// TIA Portal V20 export
DATA_BLOCK "ScaraArm3D"   // DB17, Motion_DB
// stored: InstanceOfName TO_Kinematics, OfSystemLibElement TO_Kinematics, OfSystemLibVersion 9.0
TO_Kinematics   // technology object, version 9.0
// stored: KinematicsAxis Ref J1_SCARA_Arm3D, Type TO_PositioningAxis, Index 1
// stored: KinematicsAxis Ref J3_SCARA_Arm3D, Type TO_PositioningAxis, Index 2
// stored: KinematicsAxis Ref J2_SCARA_Arm3D, Type TO_PositioningAxis, Index 3
// stored: KinematicsAxis Ref J4_SCARA_Arm3D, Type TO_PositioningAxis, Index 4
   // // inherited from TO_Object
   // VAR
   //    Tcp { ExternalWritable := 'False'; S7_SetPoint := 'True'} : TO_Struct_Kinematics_StatusKinematicsFrameTcp;
   //    Kinematics { S7_SetPoint := 'True'} : TO_Struct_Kinematics_Kinematics;
   //    KcsFrame { S7_SetPoint := 'True'} : TO_Struct_Kinematics_Frame;
   //    OcsFrame { S7_SetPoint := 'True'} : Array[1..3] of TO_Struct_Kinematics_Frame;
   //    Tool { S7_SetPoint := 'True'} : Array[1..3] of TO_Struct_Kinematics_Tool;
   //    DynamicDefaults { S7_SetPoint := 'True'} : TO_Struct_Kinematics_DynamicDefaults;
   //    DynamicLimits { S7_SetPoint := 'True'} : TO_Struct_Kinematics_DynamicLimits;
   //    Joint { S7_SetPoint := 'True'} : TO_Struct_Kinematics_Joint;
   //    AxisCoupling { S7_SetPoint := 'True'} : TO_Struct_Kinematics_AxisCoupling;
   //    MotionQueue { ExternalWritable := 'False'; S7_SetPoint := 'True'} : TO_Struct_Kinematics_MotionQueue;
   //    Transition { S7_SetPoint := 'True'} : TO_Struct_Kinematics_Transition;
   //    Override { S7_SetPoint := 'True'} : TO_Struct_Kinematics_Override;
   //    Conveyor { S7_SetPoint := 'True'} : TO_Struct_Kinematics_Conveyor;
   //    WorkspaceZone { S7_SetPoint := 'True'} : Array[1..10] of TO_Struct_Kinematics_WorkSpaceZone;
   //    KinematicsZone { S7_SetPoint := 'True'} : Array[2..10] of TO_Struct_Kinematics_KinematicsZone;
   //    StatusPath { ExternalWritable := 'False'; S7_SetPoint := 'True'} : TO_Struct_Kinematics_StatusPath;
   //    TcpInWcs { ExternalWritable := 'False'; S7_SetPoint := 'True'} : TO_Struct_Kinematics_StatusKinematicsFrameWithDynamics;
   //    TcpInOcs { ExternalWritable := 'False'; S7_SetPoint := 'True'} : Array[1..3] of TO_Struct_Kinematics_StatusKinematicsFrameWithDynamicsOcs;
   //    StatusOcsFrame { ExternalWritable := 'False'; S7_SetPoint := 'True'} : Array[1..3] of TO_Struct_Kinematics_StatusFrame;
   //    StatusKinematics { ExternalWritable := 'False'; S7_SetPoint := 'True'} : TO_Struct_Kinematics_StatusKinematics;
   //    AxesData { ExternalWritable := 'False'; S7_SetPoint := 'True'} : TO_Struct_Kinematics_AxesData;
   //    JointData { ExternalWritable := 'False'; S7_SetPoint := 'True'} : TO_Struct_Kinematics_StatusJointData;
   //    FlangeInKcs { ExternalWritable := 'False'; S7_SetPoint := 'True'} : TO_Struct_Kinematics_StatusFlangeInKcs;
   //    StatusTool { ExternalWritable := 'False'; S7_SetPoint := 'True'} : TO_Struct_Kinematics_StatusTool;
   //    StatusConveyor { ExternalWritable := 'False'; S7_SetPoint := 'True'} : Array[1..3] of TO_Struct_Kinematics_StatusConveyor;
   //    StatusWorkspaceZone { ExternalWritable := 'False'; S7_SetPoint := 'True'} : Array[1..10] of TO_Struct_Kinematics_StatusWorkSpaceZone;
   //    StatusKinematicsZone { ExternalWritable := 'False'; S7_SetPoint := 'True'} : Array[2..10] of TO_Struct_Kinematics_StatusKinematicsZone;
   //    StatusZoneMonitoring { ExternalWritable := 'False'; S7_SetPoint := 'True'} : TO_Struct_Kinematics_StatusZoneMonitoring;
   //    StatusMotionQueue { ExternalWritable := 'False'; S7_SetPoint := 'True'} : TO_Struct_Kinematics_StatusMotionQueue;
   //    KinematicsAxis { ExternalWritable := 'False'; S7_SetPoint := 'True'} : TO_Struct_Kinematics_KinematicsAxis;
   //    Units { ExternalWritable := 'False'; S7_SetPoint := 'True'} : TO_Struct_Kinematics_Units;
   //    StatusInterpreterMotion { ExternalWritable := 'False'; S7_SetPoint := 'True'} : TO_Struct_Kinematics_StatusInterpreterMotion;
   //    StatusWord { ExternalWritable := 'False'} : DWord;
   //    ErrorWord { ExternalWritable := 'False'} : DWord;
   //    ErrorDetail { ExternalWritable := 'False'; S7_SetPoint := 'True'} : TO_Struct_ErrorDetail;
   //    WarningWord { ExternalWritable := 'False'} : DWord;
   //    ControlPanel { S7_SetPoint := 'True'} : TO_Struct_Kinematics_ControlPanel;
   //    InternalToTrace { S7_SetPoint := 'True'} : Array[1..4] of TO_Struct_Internal;
   // END_VAR
BEGIN
   Kinematics.TypeOfKinematics := 10;
   Kinematics.Parameter[1] := 1028.48;
   Kinematics.Parameter[2] := 1150.0;
   Kinematics.Parameter[5] := 1200.0;
   Kinematics.Parameter[9..32] := 0.0;
   KcsFrame.x := 0.0;
   KcsFrame.y := 0.0;
   KcsFrame.z := 0.0;
   KcsFrame."a" := 0.0;
   KcsFrame."b" := 0.0;
   KcsFrame.c := 0.0;
   OcsFrame[2..3].x := 0.0;
   OcsFrame[2..3].y := 0.0;
   OcsFrame[2..3].z := 0.0;
   OcsFrame[2..3]."a" := 0.0;
   OcsFrame[1..3]."b" := 0.0;
   OcsFrame[1..3].c := 0.0;
   Tool[2..3].Frame.x := 0.0;
   Tool[2..3].Frame.y := 0.0;
   Tool[1].Frame.z := 50.0;
   Tool[2..3].Frame.z := 0.0;
   Tool[1..3].Frame."a" := 0.0;
   DynamicDefaults.Path.Velocity := 2000.0;
   DynamicDefaults.Path.Acceleration := 10000.0;
   DynamicDefaults.Path.Deceleration := 10000.0;
   DynamicDefaults.Path.Jerk := 100000.0;
   DynamicDefaults.Orientation.Velocity := 2000.0;
   DynamicDefaults.Orientation.Acceleration := 20000.0;
   DynamicDefaults.Orientation.Deceleration := 20000.0;
   DynamicDefaults.Orientation.Jerk := 1000000.0;
   DynamicDefaults.DynamicAdaption := 1;
   DynamicDefaults.MoveDirect.VelocityFactor := 0.5;
   DynamicDefaults.MoveDirect.AccelerationFactor := 0.5;
   DynamicDefaults.MoveDirect.DecelerationFactor := 0.5;
   DynamicDefaults.MoveDirect.JerkFactor := 0.5;
   DynamicLimits.Path.Velocity := 3000.0;
   DynamicLimits.Path.Acceleration := 100000.0;
   DynamicLimits.Path.Deceleration := 100000.0;
   DynamicLimits.Orientation.Velocity := 2200.0;
   DynamicLimits.Orientation.Acceleration := 20000.0;
   DynamicLimits.Orientation.Deceleration := 20000.0;
   DynamicLimits.Orientation.Jerk := 1000000.0;
   Override.Velocity := 62.0;
   WorkspaceZone[1].Active := true;
   WorkspaceZone[2..10].Active := false;
   WorkspaceZone[1].Valid := true;
   WorkspaceZone[2..10].Valid := false;
   WorkspaceZone[2..10]."Type" := 1;
   WorkspaceZone[1..10].ReferenceSystem := 0;
   WorkspaceZone[2..10].Frame.x := 0.0;
   WorkspaceZone[2..10].Frame.y := 0.0;
   WorkspaceZone[1].Frame.z := -100.0;
   WorkspaceZone[2..10].Frame.z := 0.0;
   WorkspaceZone[1..10].Frame."a" := 0.0;
   WorkspaceZone[1..10].Frame."b" := 0.0;
   WorkspaceZone[1..10].Frame.c := 0.0;
   WorkspaceZone[1].Geometry."Type" := 2;
   WorkspaceZone[2..10].Geometry."Type" := 0;
   WorkspaceZone[1].Geometry.Parameter[1] := 2500.0;
   WorkspaceZone[1].Geometry.Parameter[2] := 2000.0;
   WorkspaceZone[1].Geometry.Parameter[3] := 500.0;
   WorkspaceZone[2].Geometry.Parameter[1..3] := 500.0;
   WorkspaceZone[3].Geometry.Parameter[1..3] := 500.0;
   WorkspaceZone[4].Geometry.Parameter[1..3] := 500.0;
   WorkspaceZone[5].Geometry.Parameter[1..3] := 500.0;
   WorkspaceZone[6].Geometry.Parameter[1..3] := 500.0;
   WorkspaceZone[7].Geometry.Parameter[1..3] := 500.0;
   WorkspaceZone[8].Geometry.Parameter[1..3] := 500.0;
   WorkspaceZone[9].Geometry.Parameter[1..3] := 500.0;
   WorkspaceZone[10].Geometry.Parameter[1..3] := 500.0;
   KinematicsZone[3..10].Active := false;
   KinematicsZone[3..10].Valid := false;
   KinematicsZone[2..10].ReferenceSystem := 0;
   KinematicsZone[2..10].Frame.x := 0.0;
   KinematicsZone[2..10].Frame.y := 0.0;
   KinematicsZone[2..10].Frame.z := 0.0;
   KinematicsZone[2..10].Frame."a" := 0.0;
   KinematicsZone[2..10].Frame."b" := 0.0;
   KinematicsZone[2..10].Frame.c := 0.0;
   KinematicsZone[2].Geometry."Type" := 2;
   KinematicsZone[3..10].Geometry."Type" := 0;
   KinematicsZone[2].Geometry.Parameter[1] := 5000.0;
   KinematicsZone[2].Geometry.Parameter[2] := 3000.0;
   KinematicsZone[2].Geometry.Parameter[3] := 5000.0;
   KinematicsZone[3].Geometry.Parameter[1..3] := 500.0;
   KinematicsZone[4].Geometry.Parameter[1..3] := 500.0;
   KinematicsZone[5].Geometry.Parameter[1..3] := 500.0;
   KinematicsZone[6].Geometry.Parameter[1..3] := 500.0;
   KinematicsZone[7].Geometry.Parameter[1..3] := 500.0;
   KinematicsZone[8].Geometry.Parameter[1..3] := 500.0;
   KinematicsZone[9].Geometry.Parameter[1..3] := 500.0;
   KinematicsZone[10].Geometry.Parameter[1..3] := 500.0;
   ControlPanel.Input.TimeOut := 2000.0;
   ControlPanel.Input.EsLifeSign := 0;
   ControlPanel.Input.Command[1..2].ReqCounter := 0;
   ControlPanel.Input.Command[1..2]."Type" := 0;
   ControlPanel.Input.Command[1].Position[1..4] := 0.0;
   ControlPanel.Input.Command[2].Position[1..4] := 0.0;
   ControlPanel.Input.Command[1].Velocity[1..2] := 0.0;
   ControlPanel.Input.Command[2].Velocity[1..2] := 0.0;
   ControlPanel.Input.Command[1].Acceleration[1..2] := 0.0;
   ControlPanel.Input.Command[2].Acceleration[1..2] := 0.0;
   ControlPanel.Input.Command[1].Deceleration[1..2] := 0.0;
   ControlPanel.Input.Command[2].Deceleration[1..2] := 0.0;
   ControlPanel.Input.Command[1].Jerk[1..2] := 0.0;
   ControlPanel.Input.Command[2].Jerk[1..2] := 0.0;
   ControlPanel.Input.Command[1].Param[1..9] := 0.0;
   ControlPanel.Input.Command[2].Param[1..9] := 0.0;
   ControlPanel.Input.Command[1..2].CoordinateSystem := 0;
   ControlPanel.Input.Command[1..2].ToolNumber := 0;
   InternalToTrace[1..4].Id := 0;
   InternalToTrace[1..4].Value := 0.0;
   Kinematics.TypeOfKinematics := 10;
END_DATA_BLOCK
